//{attribute 'qualified_only'}
{attribute 'strict'}
TYPE eMC_State_Machine :
(
		MC_Init 			:= 0 ,
		MC_Power 			:= 1 ,
		MC_Ready 			:= 2 ,
		MC_Home 			:= 3 ,
		MC_ManualMovement 	:= 4 ,
		MC_AutoMovement 	:= 5 ,
		MC_Error 			:= 6 ,
		MC_Reset 			:= 7

);
END_TYPE

(* stored: Version 1.1.0.1, ProductVersion 3.1.4024.3
   EnumerationTextList eMC_State_Machine: Id {7e01dfd9-388f-4b3f-897d-3afc2396dd05} *)
